// TIA Portal V19 export
TYPE "LUC_typeStateMachineConfiguration"
TITLE = LUC_typeStateMachineConfiguration
// Configuration of the state machine
// stored: Access Published
   STRUCT
      enableModes : "LUC_typeModeConfiguration";
      enableStates : Array[0.."LPMLV2022_MAX_MODES_UPPER_LIM"] of "LUC_typeStateConfiguration";
      enableModeTransitions : Array[0.."LPMLV2022_MAX_MODES_UPPER_LIM"] of "LUC_typeModeTransitionConfiguration";
      enableHoldCommand : "LUC_typeHoldCommandConfiguration";
      enableCompleteCommand : "LUC_typeCompleteCommandConfiguration";
   END_STRUCT;
   // // enableStates[0] : Mode_Invalid, Not used
   // // enableStates[1] : For mode production
   // // enableStates[2] : For mode maintenance
   // // enableStates[3] : For mode manual
   // // enableStates[4] : For userMode01
   // // enableStates[5] : For userMode02
   // // enableStates[6] : For userMode03
   // // enableStates[7] : For userMode04
   // // enableStates[8] : For userMode05
   // enableStates[3].starting := false;
   // enableStates[2..3].suspended := false;
   // enableStates[3].holding := false;
   // enableStates[3].held := false;
   // enableStates[3].unholding := false;
   // enableStates[2..3].suspending := false;
   // enableStates[2..3].unsuspending := false;
   // enableStates[2..3].completing := false;
   // enableStates[2..3].completed := false;
   // // enableModeTransitions[0] : Mode_Invalid, Not used
   // // enableModeTransitions[1] : For mode production
   // // enableModeTransitions[2] : For mode maintenance
   // // enableModeTransitions[3] : For mode manual
   // // enableModeTransitions[4] : For userMode01
   // // enableModeTransitions[5] : For userMode02
   // // enableModeTransitions[6] : For userMode03
   // // enableModeTransitions[7] : For userMode04
   // // enableModeTransitions[8] : For userMode05
END_TYPE
